FUNCTION ReadModusTime : Time
VAR_INPUT
END_VAR
VAR
	i: INT;
	modbusTime: ModbusUnion;
END_VAR


i:= GVL.nOutputRegisterIndex;

modbusTime.longValue:= GVL.mb_Output_Registers[i+0] * 1000;

GVL.nOutputRegisterIndex:= i + 0;


ReadModusTime := modbusTime.timeValue;

END_FUNCTION

(* stored: Version 1.1.0.1, ProductVersion 3.1.4024.12
   POU ReadModusTime: Id {2f3a2243-5d01-4e49-848f-77986b00727c}, SpecialFunc None *)
